% RSLogix 500 project ERROR FLASHER_BAK039.RSS, saved by version 10.00.00.00 %
PROJECT "UNTITLED"    % processor: Bul.1763 MicroLogix 1100 Series B %

PROGRAM FILES
  LAD 2   3 rungs
  LAD 4 "ERR"  6 rungs  % Error Flasher %

DATA FILES
  O0 OUTPUT  4 elements
  I1 INPUT  6 elements
  S2 STATUS  66 elements
  B3 BINARY  12 elements
  T4 TIMER  17 elements
  C5 COUNTER  12 elements
  R6 CONTROL  1 elements
  N7 INTEGER  13 elements
  F8 FLOAT  1 elements

LADDER 2
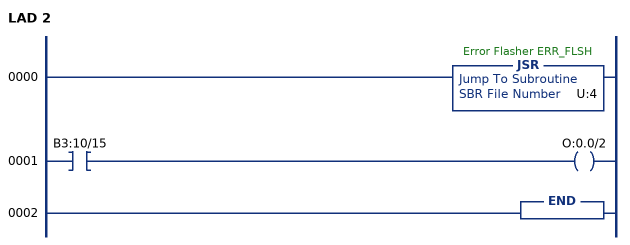
% Rung: 0 %
SOR JSR U:4 EOR
%   U:4  ERR_FLSH  "Error Flasher" %
% Rung: 1 %
SOR XIC B3:10/15 OTE O:0.0/2 EOR
% Rung: 2 %
SOR END EOR

LADDER 4 "ERR"    % Error Flasher %
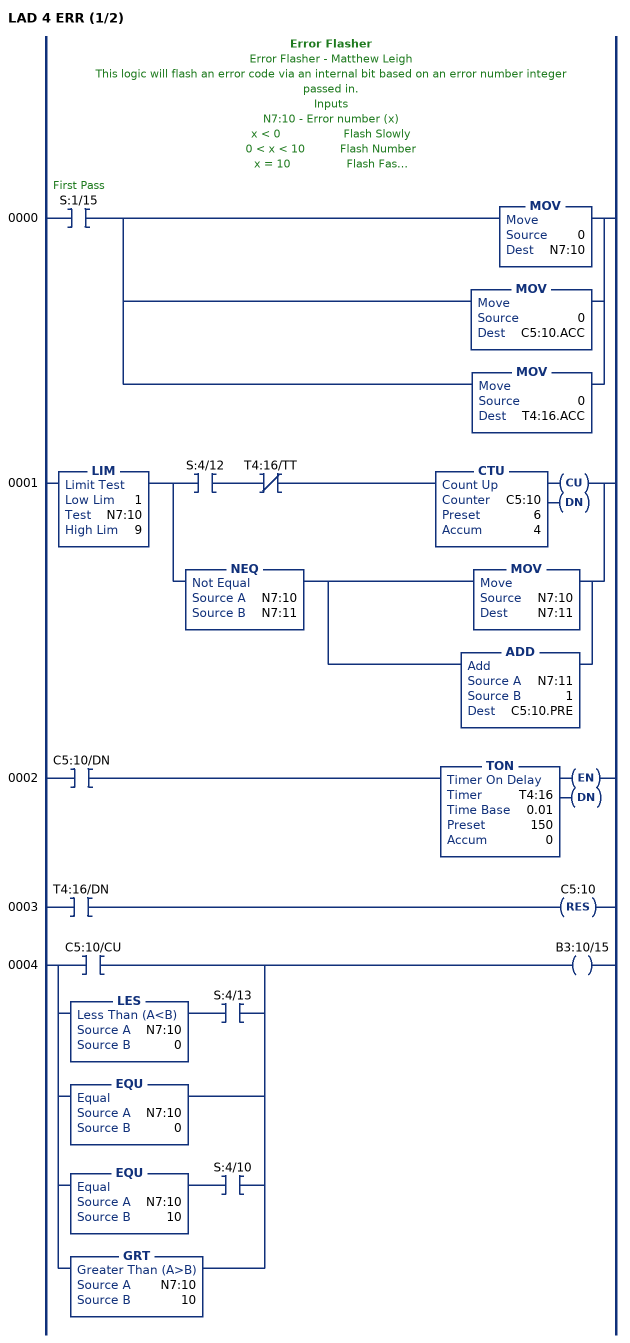
% Rung: 0 %
% TITLE: Error Flasher %
% Error Flasher - Matthew Leigh
% This logic will flash an error code via an internal bit based on an error number integer passed in.
% 
% Inputs
%    N7:10 - Error number (x)
%       x < 0                  Flash Slowly
%       0 < x < 10          Flash Number
%       x = 10                Flash Fast
%       x = 0 or x > 10   On Solid
% 
% Outputs
%    B3:10/15 - Flashing bit %
SOR XIC S:1/15 BST MOV 0 N7:10 NXB MOV 0 C5:10.ACC NXB MOV 0 T4:16.ACC BND EOR
%   S:1/15  "First Pass" %
% Rung: 1 %
SOR LIM 1 N7:10 9 BST XIC S:4/12 XIO T4:16/TT CTU C5:10 6 4 NXB NEQ N7:10 N7:11 BST MOV N7:10 N7:11 NXB ADD N7:11 1 C5:10.PRE BND BND EOR
% Rung: 2 %
SOR XIC C5:10/DN TON T4:16 0.01 150 0 EOR
% Rung: 3 %
SOR XIC T4:16/DN RES C5:10 EOR
% Rung: 4 %
SOR BST XIC C5:10/CU NXB LES N7:10 0 XIC S:4/13 NXB EQU N7:10 0 NXB EQU N7:10 10 XIC S:4/10 NXB GRT N7:10 10 BND OTE B3:10/15 EOR

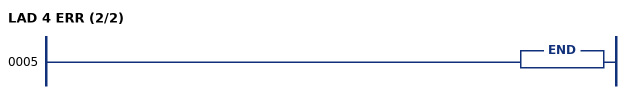
% Rung: 5 %
SOR END EOR

OTHER DOCUMENTED ADDRESSES
  B3:0/0  ERR  "Error Active"
  B3:0/1  ONES
  B3:0/2  TEENS
  B3:0/3  TWENTIES  "Twenties"
  B3:10/14  ERR_RNG  "In Error Range"
  N7:0  ERR_NUM  "Error Number"
  N7:1  ONES_PLC  "Ones Place"
  N7:2  TENS_PLC  "Tens Place"

DATA TABLE (non-zero values as saved)
DATA B3
% B3:0 % 0X0005 0X0000 0X0000 0X0000 0X0000 0X0000 0X0000 0X0000 0X0000 0X0000
% B3:10 % 0XC000 0X0000
DATA T4
% .PRE .ACC %
% T4:0 % 32767 0
% T4:15 % 150 150
% T4:16 % 150 0
DATA C5
% .PRE .ACC %
% C5:10 % 6 4
% C5:11 % 6 5
DATA N7
% N7:0 % 0 2 1 0 0 0 0 0 0 0
% N7:10 % 20 5 0
